FUNCTION_BLOCK FB_EmptyBlock_1
VAR_INPUT
END_VAR
VAR_OUTPUT
END_VAR
VAR
	value : BOOL;
END_VAR

END_FUNCTION_BLOCK

(* stored: Version 1.1.0.1, ProductVersion 3.1.4024.12
   POU FB_EmptyBlock_1: Id {09b56bc8-3db5-44a1-8c7e-13070912ab68}, SpecialFunc None *)
